// TIA Portal V19 export
TYPE "TetraPakV70_IO"
TITLE = TP_V70_10_IO
// DEVICEID : 10
//  VENDOR : IFM on behalf of Tetra Pak
//  DATE: 27.12.2023 
// 
//  Comment : TP V70 IO Interface
   STRUCT
      IN_Address : Int;   // First Byte address of 4 byte address space
      IN_Pulse : Bool;   // Trigger one clean pulse on SV_1
      IN_SV_1 : Bool;   // Trigger solenoid valve 1 for main valve activation
      IN_Wink : Bool;   // Visual indictation for locating the unit
      IN_SV_2 : Bool;   // Trigger solenoid valve 2 for upper seat lift activation
      IN_SV_3 : Bool;   // Trigger solenoid valve 3 for lower seat push activation
      IN_Burst : Bool;   // Enable burst clean
      OUT_LSP : Bool;   // Lower Seat Push energised position
      OUT_USL : Bool;   // Upper Seat Lift energised position
      OUT : Struct
         ValvePosition : Real;   // Current Valve Position (0 - 1060 * 0.1)
         ErrorStatus : Byte;   // See Block Comment
         ValveState : Bool;   // Current Valve State
         Main : Bool;   // Main energised position
         DE_EN : Bool;   // De-energised
         O_DI4 : Bool;   // Output signal status Pin 4
         O_DI2 : Bool;   // Output signal status Pin 2
         O_DA : Bool;   // Output device recognised
         O_DE : Bool;   // Output device error event has appeared
         O_PQ : Bool;   // Output port qualifer proces data valid
      END_STRUCT;
      IN_OUT : Struct
         HMI_INFO : Int;
         HMI_CMD : Int;
      END_STRUCT;
   END_STRUCT;
END_TYPE
